{attribute 'linkalways'} 
{attribute 'no_explicit_call' := 'This FB is a CLASS and must be accessed using methods or properties'}
{attribute 'enable_dynamic_creation'}
FUNCTION_BLOCK FINAL SUB_SINT EXTENDS Node
VAR
	in1 : _SINT(0);
	in2 : _SINT(0);
	out : _SINT(0);
END_VAR

METHOD PUBLIC Clone : I_Node
VAR
	pNode : POINTER TO SUB_SINT;
END_VAR
pNode := __NEW(SUB_SINT);
Clone := pNode^;
END_METHOD

METHOD FB_init : BOOL
VAR_INPUT
	bInitRetains : BOOL; // if TRUE, the retain variables are initialized (warm start / cold start)
	bInCopyCode : BOOL;  // if TRUE, the instance afterwards gets moved into the copy code (online change)
END_VAR
AddInput('in1',THIS^.in1);
AddInput('in2',THIS^.in2);
AddOutput('out', THIS^.out);
END_METHOD

METHOD PROTECTED OnExecute
VAR
END_VAR
out.Value := in1.Value - in2.Value;
END_METHOD

END_FUNCTION_BLOCK

(* stored: Version 1.1.0.1, ProductVersion 3.1.4024.15
   POU SUB_SINT: Id {eb62f237-bd65-4295-a75d-a807e12c12d5}, SpecialFunc None
   Folder Constructor: Id {5d37d59f-84d8-47bb-a435-552cb87bc540}
   Method Clone: Id {7bbe17c7-64c3-4655-9177-dd8ed08d7953}
   Method FB_init: Id {a0ae15f3-bce4-40a9-8b0c-602624f7ac55}
   Method OnExecute: Id {42d23b97-b81d-4435-87b8-bdbb94bd6516} *)
